// LS Electric XG5000 project: 63_3_A
// PLC NewPLC
// module base 0 slot 0: 입출력 모듈:XBC-DR20S (DC 24V 입력 12점, 릴레이 출력 8점)

PROGRAM NewProgram (task: 스캔 프로그램)

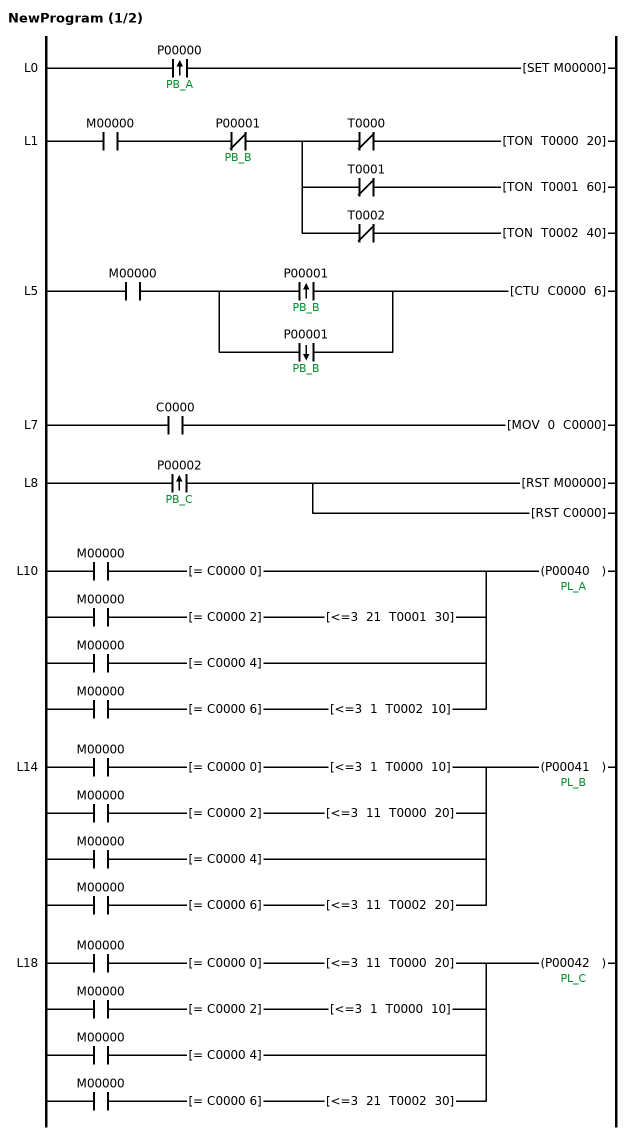
; L0
LOADP     P00000	// PB_A
SET       M00000
; L1
LOAD      M00000
AND NOT   P00001	// PB_B
MPUSH
AND NOT   T0000
TON       T0000 20
MLOAD
AND NOT   T0001
TON       T0001 60
MPOP
AND NOT   T0002
TON       T0002 40
; L5
LOAD      M00000
LOADP     P00001	// PB_B
ORN       P00001	// PB_B
AND LOAD
CTU       C0000 6
; L7
LOAD      C0000
MOV       0 C0000
; L8
LOADP     P00002	// PB_C
RST       M00000
RST       C0000
; L10
LOAD      M00000
AND=      C0000 0
LOAD      M00000
AND=      C0000 2
AND<=3    21 T0001 30
OR LOAD
LOAD      M00000
AND=      C0000 4
OR LOAD
LOAD      M00000
AND=      C0000 6
AND<=3    1 T0002 10
OR LOAD
OUT       P00040	// PL_A
; L14
LOAD      M00000
AND=      C0000 0
AND<=3    1 T0000 10
LOAD      M00000
AND=      C0000 2
AND<=3    11 T0000 20
OR LOAD
LOAD      M00000
AND=      C0000 4
OR LOAD
LOAD      M00000
AND=      C0000 6
AND<=3    11 T0002 20
OR LOAD
OUT       P00041	// PL_B
; L18
LOAD      M00000
AND=      C0000 0
AND<=3    11 T0000 20
LOAD      M00000
AND=      C0000 2
AND<=3    1 T0000 10
OR LOAD
LOAD      M00000
AND=      C0000 4
OR LOAD
LOAD      M00000
AND=      C0000 6
AND<=3    21 T0002 30
OR LOAD
OUT       P00042	// PL_C

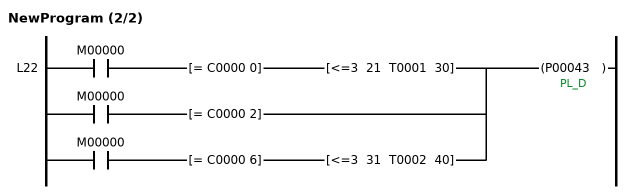
; L22
LOAD      M00000
AND=      C0000 0
AND<=3    21 T0001 30
LOAD      M00000
AND=      C0000 2
OR LOAD
LOAD      M00000
AND=      C0000 6
AND<=3    31 T0002 40
OR LOAD
OUT       P00043	// PL_D

VARIABLES AND COMMENTS (devices not used above)
P00044	BIT	PL_E